TYPE ST_Solvents :
STRUCT
	Solvent_ID 		: INT;
	solventName1 	: STRING(100);
	solventName2 	: STRING(100);
	solventName3 	: STRING(100);
	solventName4 	: STRING(100);
	density1 		: STRING(100);
	density2 		: STRING(100);
	density3 		: STRING(100);
	density4 		: STRING(100);
	addedBy 		: STRING(100);
	addedDate 		: STRING(100);
END_STRUCT
END_TYPE

(* stored: Version 1.1.0.1, ProductVersion 3.1.4024.15
   DUT ST_Solvents: Id {50b8591c-eb8c-487b-abc8-4b9d47f65a87} *)
